// TIA Portal V19 export
TYPE "typeTotal64REAL"
   STRUCT
      preset { S7_SetPoint := 'True'} : Real;   // Preset quantity to add with each pulse
      precision { S7_SetPoint := 'True'} : USInt;   // Maximum decimal precision
      output : LReal;   // Totalizer's output
      reset : Bool;   // Null totalizer
   END_STRUCT;
END_TYPE
